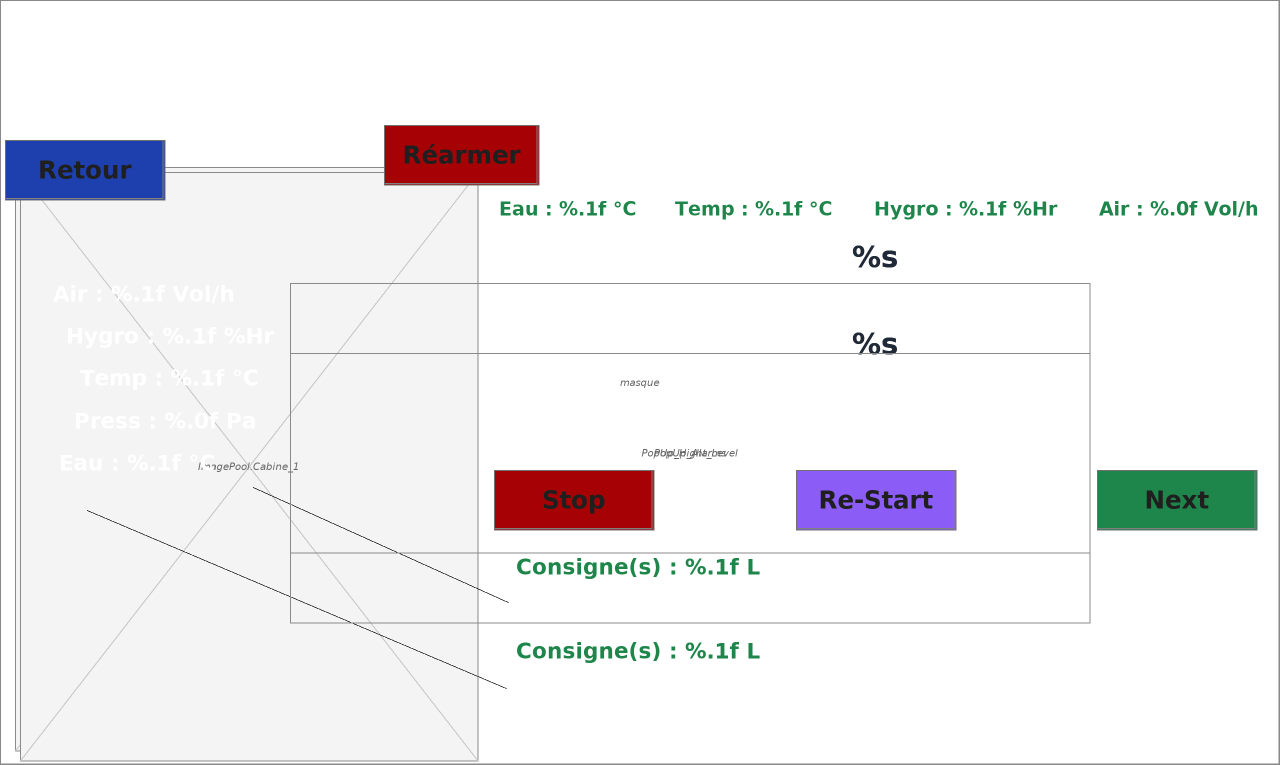
VISUALIZATION Recet_EnCours  // 1280x765
    Frame (0,0 1280x765)
        shows masque()
    Group (494,149 763x386), invisible if: NOT Mode_Cabine_Automatique
        Button (0,321 160x60), "Stop"
            OnMouseDown: toggle Reset_Mode_Auto
        Rectangle (81,0 615x49), "MODE RECETTE EN COURS", invisible if: GVL_Visu.On_Off_Anim
        Button (603,321 160x60), "Next", invisible if: NOT Condi_Affich_Etape_Suiv
            OnMouseDown: toggle Valid_Texte
        Button (302,321 160x60), "Re-Start", invisible if: NOT Statut_Pause_Force
            OnMouseDown: toggle Bp_Pause
    Image (15,167 463x584), image: ImagePool.Cabine-2
    Polygon (42,662) (181,704) (321,739) (395,704) (468,662), colour variable: GVL_Visu.Couleur_Cabine
    Polygon (44,662) (42,246) (323,185) (465,254) (467,662), colour variable: GVL_Visu.Couleur_Cabine
    Image (20,172 458x589), image: ImagePool.Cabine_1
        OnMouseDown: OpenDialog Dialog=Actionneurs, OpenModal=True, OpenCentered=True
    Group (834,583 431x127), invisible if: NOT GVL_Visu.Visu_Tempo
        Rectangle (0,0 319x42), "Heure(s) restante(s) :"
        Rectangle (319,0 112x42), "%.0f hrs", text variable: Temp_Restant_Heure
        Rectangle (0,85 319x42), "Seconde(s) restante(s) :"
        Rectangle (319,85 112x42), "%.0f sec", text variable: Temp_Restant_Seconde
        Rectangle (0,42 319x42), "Minute(s) restante(s) :"
        Rectangle (319,42 112x42), "%.0f min", text variable: Temp_Restant_Minute
    Button (5,140 160x60), "Retour", invisible if: Mode_Cabine_Automatique
        OnMouseDown: change screen: menu
    Rectangle (496,402 176x42), "Etape : %d /", text variable: Numero_Etape_Actuel
    Rectangle (676,402 112x42), "%d", text variable: Nbre_Etape_Totale
    Rectangle (1075,402 176x42), "Mode N°%.0f", text variable: Numero_Mode_Actuel
    Group (494,226 763x62)
        RoundedRectangle (0,0 763x62)
        Rectangle (0,0 763x62), "%s", text variable: Tab_Nom_Recette[1,0], invisible if: VisuElems.CURRENTLANGUAGE = 'en'
        Rectangle (0,0 763x62), "%s", text variable: Tab_Nom_Recette[2,0], invisible if: VisuElems.CURRENTLANGUAGE = 'fr'
    Group (494,287 763x114)
        RoundedRectangle (0,0 763x114)
        Rectangle (0,0 763x114), "%s", text variable: Lecture_Texte_Choisi_FR, invisible if: VisuElems.CURRENTLANGUAGE = 'en'
        Rectangle (0,0 763x114), "%s", text variable: Lecture_Texte_Choisi_ENG, invisible if: VisuElems.CURRENTLANGUAGE = 'fr'
    Group (496,192 777x34)
        Rectangle (0,0 171x34), "Eau : %.1f °C", text variable: n3_Regul_Temp_EauMitig.SetPoint_PID_Temp_EM, invisible if: NOT a5_Ecriture_InterCom.Dmd_Mise_En_Temp
        Rectangle (176,0 196x34), "Temp : %.1f °C", text variable: Lect_Cons_Temperature_Cabine, invisible if: NOT RS_MEnCond.Q1
        Rectangle (375,0 233x34), "Hygro : %.1f %Hr", text variable: Lect_Cons_Hygrometrie_Cabine, invisible if: NOT RS_MEnCond.Q1
        Rectangle (600,0 177x34), "Air : %.0f Vol/h", text variable: Cons_Actionneur_Registre_Souf_Volh
    Group (823,709 442x42), invisible if: NOT GVL_Visu.Visu_ChasseEau
        Rectangle (0,0 319x42), "Chasse(s) restante(s) :"
        Rectangle (319,0 73x42), "%.0f /", text variable: Nbre_Chasse_EnCours
        Rectangle (385,0 57x42), "%.0f", text variable: Nbre_Chasse_Total
    Group (253,487 602x140), invisible if: NOT GVL_Visu.Visu_VolEau_Douche
        Line (0,0) (255,115)
        Rectangle (260,98 342x42), "Volume d'eau : %.1f L", text variable: Lect_Volume_Eau_Douche
        Rectangle (260,63 342x34), "Consigne(s) : %.1f L", text variable: Cons_Volume_Eau_Douche_Actuel
    Group (87,510 768x200), invisible if: NOT GVL_Visu.Visu_VolEau_Lavabo
        Line (0,0) (419,178)
        Rectangle (426,158 342x42), "Volume d'eau : %.1f L", text variable: Lect_Volume_Eau_Lavabo
        Rectangle (426,124 342x34), "Consigne(s) : %.1f L", text variable: Cons_Volume_Eau_Lavabo_Actuel
    Button (384,125 155x60), "Réarmer", invisible if: NOT Condi_Affich_Rearm
        OnMouseDown: toggle Cmd_Rearmement
    Group (50,273 319x211)
        Rectangle (13,42 292x42), "Hygro : %.1f %Hr", text variable: Tab_MES_Sonde_Hygro_Amb.R_MesCor
        Rectangle (27,84 292x42), "Temp : %.1f °C", text variable: Tab_MES_Sonde_Temp_Amb.R_MesCor
        Rectangle (0,0 292x42), "Air : %.1f Vol/h", text variable: MES_Debit_Volh_Soufflage, invisible if: TRUE
        Rectangle (21,127 292x42), "Press : %.0f Pa", text variable: Tab_MES_Sonde_Press_Cab.R_MesCor
        Rectangle (6,169 292x42), "Eau : %.1f °C", text variable: MES_Temp_Eau_Mitige_General
    Rectangle (513,711 292x42), "Débit : %.1f l/min", text variable: GVL_Visu.Visu_Mes_Debit_Eau, invisible if: NOT GVL_Visu.Visu_Debit_Eau
    Group (290,283 800x340)
        Frame (0,0 800x340), invisible if: NOT GVL_Visu.Affichage_PopUp_Alarm
            shows PopUp_Alarms()
        Frame (0,70 800x200), invisible if: NOT GVL_Visu.Affichage_PopUp_HightLevel
            shows PopUp_Hight_Level()
END_VISUALIZATION

(* stored: Version 1.1.0.1, ProductVersion 3.1.4024.16
   Visu Recet_EnCours: Id {385c87ca-027e-4b3d-be96-c59542f655f1} *)
